// TIA Portal V20 export
FUNCTION "Map01" : Void   // FC126, LAD
// stored: Namespace Unit1, SetENOAutomatically false
   VAR_TEMP   // added for the SCL form of the ladder/FBD networks
      _w1 : Bool;
   END_VAR
BEGIN

REGION Network 1: Autocycle Running
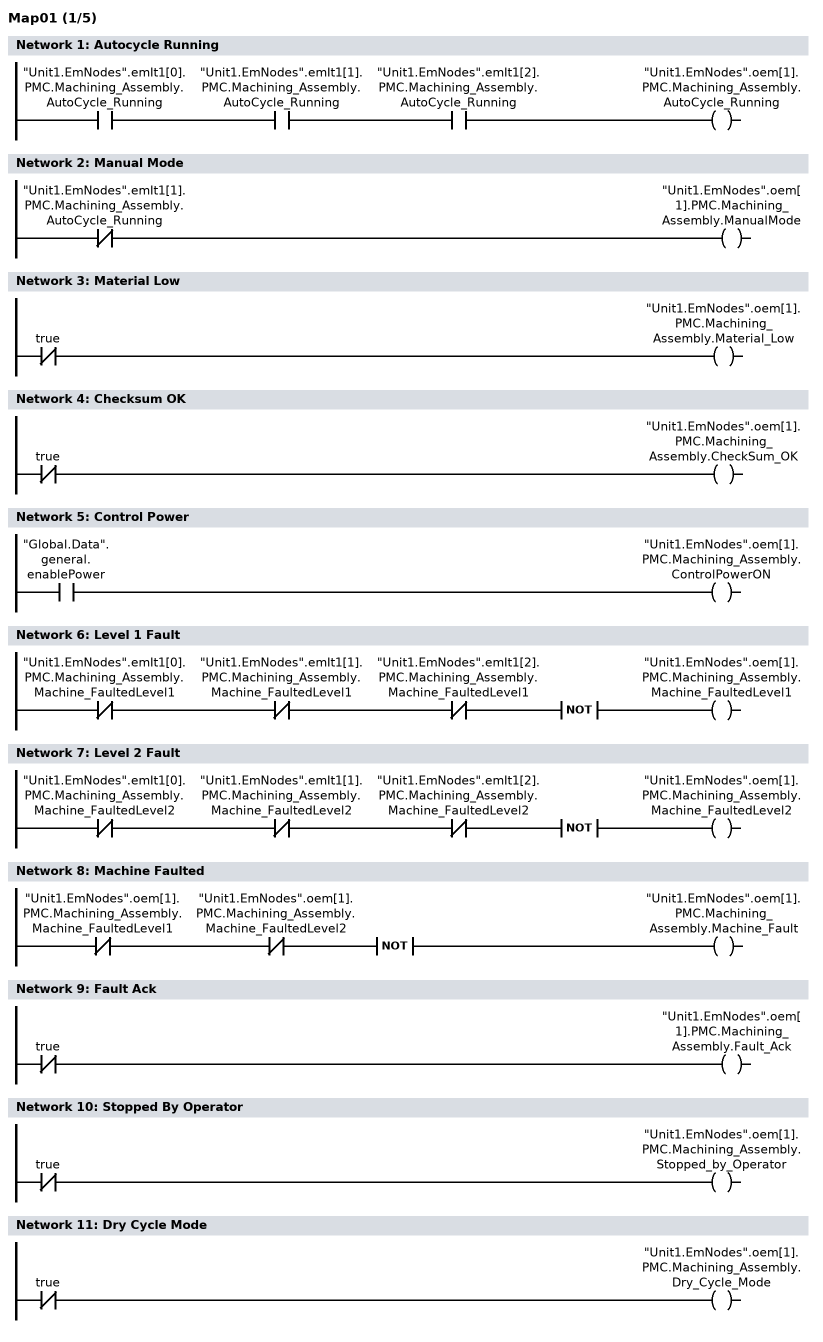
   RUNG wire#powerrail
      Contact( "Unit1.EmNodes".emIt1[0].PMC.Machining_Assembly.AutoCycle_Running )
      Contact( "Unit1.EmNodes".emIt1[1].PMC.Machining_Assembly.AutoCycle_Running )
      Contact( "Unit1.EmNodes".emIt1[2].PMC.Machining_Assembly.AutoCycle_Running )
      Coil( "Unit1.EmNodes".oem[1].PMC.Machining_Assembly.AutoCycle_Running )
   END_RUNG
   // the same network as SCL:
   "Unit1.EmNodes".oem[1].PMC.Machining_Assembly.AutoCycle_Running := "Unit1.EmNodes".emIt1[0].PMC.Machining_Assembly.AutoCycle_Running AND "Unit1.EmNodes".emIt1[1].PMC.Machining_Assembly.AutoCycle_Running AND "Unit1.EmNodes".emIt1[2].PMC.Machining_Assembly.AutoCycle_Running;
END_REGION

REGION Network 2: Manual Mode
   RUNG wire#powerrail
      I_Contact( "Unit1.EmNodes".emIt1[1].PMC.Machining_Assembly.AutoCycle_Running )
      Coil( "Unit1.EmNodes".oem[1].PMC.Machining_Assembly.ManualMode )
   END_RUNG
   // the same network as SCL:
   "Unit1.EmNodes".oem[1].PMC.Machining_Assembly.ManualMode := NOT "Unit1.EmNodes".emIt1[1].PMC.Machining_Assembly.AutoCycle_Running;
END_REGION

REGION Network 3: Material Low
   RUNG wire#powerrail
      I_Contact( true )
      Coil( "Unit1.EmNodes".oem[1].PMC.Machining_Assembly.Material_Low )
   END_RUNG
   // the same network as SCL:
   "Unit1.EmNodes".oem[1].PMC.Machining_Assembly.Material_Low := NOT true;
END_REGION

REGION Network 4: Checksum OK
   RUNG wire#powerrail
      I_Contact( true )
      Coil( "Unit1.EmNodes".oem[1].PMC.Machining_Assembly.CheckSum_OK )
   END_RUNG
   // the same network as SCL:
   "Unit1.EmNodes".oem[1].PMC.Machining_Assembly.CheckSum_OK := NOT true;
END_REGION

REGION Network 5: Control Power
   RUNG wire#powerrail
      Contact( "Global.Data".general.enablePower )
      Coil( "Unit1.EmNodes".oem[1].PMC.Machining_Assembly.ControlPowerON )
   END_RUNG
   // the same network as SCL:
   "Unit1.EmNodes".oem[1].PMC.Machining_Assembly.ControlPowerON := "Global.Data".general.enablePower;
END_REGION

REGION Network 6: Level 1 Fault
   RUNG wire#powerrail
      I_Contact( "Unit1.EmNodes".emIt1[0].PMC.Machining_Assembly.Machine_FaultedLevel1 )
      I_Contact( "Unit1.EmNodes".emIt1[1].PMC.Machining_Assembly.Machine_FaultedLevel1 )
      I_Contact( "Unit1.EmNodes".emIt1[2].PMC.Machining_Assembly.Machine_FaultedLevel1 )
      Not()
      Coil( "Unit1.EmNodes".oem[1].PMC.Machining_Assembly.Machine_FaultedLevel1 )
   END_RUNG
   // the same network as SCL:
   "Unit1.EmNodes".oem[1].PMC.Machining_Assembly.Machine_FaultedLevel1 := NOT (NOT "Unit1.EmNodes".emIt1[0].PMC.Machining_Assembly.Machine_FaultedLevel1 AND NOT "Unit1.EmNodes".emIt1[1].PMC.Machining_Assembly.Machine_FaultedLevel1 AND NOT "Unit1.EmNodes".emIt1[2].PMC.Machining_Assembly.Machine_FaultedLevel1);
END_REGION

REGION Network 7: Level 2 Fault
   RUNG wire#powerrail
      I_Contact( "Unit1.EmNodes".emIt1[0].PMC.Machining_Assembly.Machine_FaultedLevel2 )
      I_Contact( "Unit1.EmNodes".emIt1[1].PMC.Machining_Assembly.Machine_FaultedLevel2 )
      I_Contact( "Unit1.EmNodes".emIt1[2].PMC.Machining_Assembly.Machine_FaultedLevel2 )
      Not()
      Coil( "Unit1.EmNodes".oem[1].PMC.Machining_Assembly.Machine_FaultedLevel2 )
   END_RUNG
   // the same network as SCL:
   "Unit1.EmNodes".oem[1].PMC.Machining_Assembly.Machine_FaultedLevel2 := NOT (NOT "Unit1.EmNodes".emIt1[0].PMC.Machining_Assembly.Machine_FaultedLevel2 AND NOT "Unit1.EmNodes".emIt1[1].PMC.Machining_Assembly.Machine_FaultedLevel2 AND NOT "Unit1.EmNodes".emIt1[2].PMC.Machining_Assembly.Machine_FaultedLevel2);
END_REGION

REGION Network 8: Machine Faulted
   RUNG wire#powerrail
      I_Contact( "Unit1.EmNodes".oem[1].PMC.Machining_Assembly.Machine_FaultedLevel1 )
      I_Contact( "Unit1.EmNodes".oem[1].PMC.Machining_Assembly.Machine_FaultedLevel2 )
      Not()
      Coil( "Unit1.EmNodes".oem[1].PMC.Machining_Assembly.Machine_Fault )
   END_RUNG
   // the same network as SCL:
   "Unit1.EmNodes".oem[1].PMC.Machining_Assembly.Machine_Fault := NOT (NOT "Unit1.EmNodes".oem[1].PMC.Machining_Assembly.Machine_FaultedLevel1 AND NOT "Unit1.EmNodes".oem[1].PMC.Machining_Assembly.Machine_FaultedLevel2);
END_REGION

REGION Network 9: Fault Ack
   RUNG wire#powerrail
      I_Contact( true )
      Coil( "Unit1.EmNodes".oem[1].PMC.Machining_Assembly.Fault_Ack )
   END_RUNG
   // the same network as SCL:
   "Unit1.EmNodes".oem[1].PMC.Machining_Assembly.Fault_Ack := NOT true;
END_REGION

REGION Network 10: Stopped By Operator
   RUNG wire#powerrail
      I_Contact( true )
      Coil( "Unit1.EmNodes".oem[1].PMC.Machining_Assembly.Stopped_by_Operator )
   END_RUNG
   // the same network as SCL:
   "Unit1.EmNodes".oem[1].PMC.Machining_Assembly.Stopped_by_Operator := NOT true;
END_REGION

REGION Network 11: Dry Cycle Mode
   RUNG wire#powerrail
      I_Contact( true )
      Coil( "Unit1.EmNodes".oem[1].PMC.Machining_Assembly.Dry_Cycle_Mode )
   END_RUNG
   // the same network as SCL:
   "Unit1.EmNodes".oem[1].PMC.Machining_Assembly.Dry_Cycle_Mode := NOT true;
END_REGION

REGION Network 12: Blocked
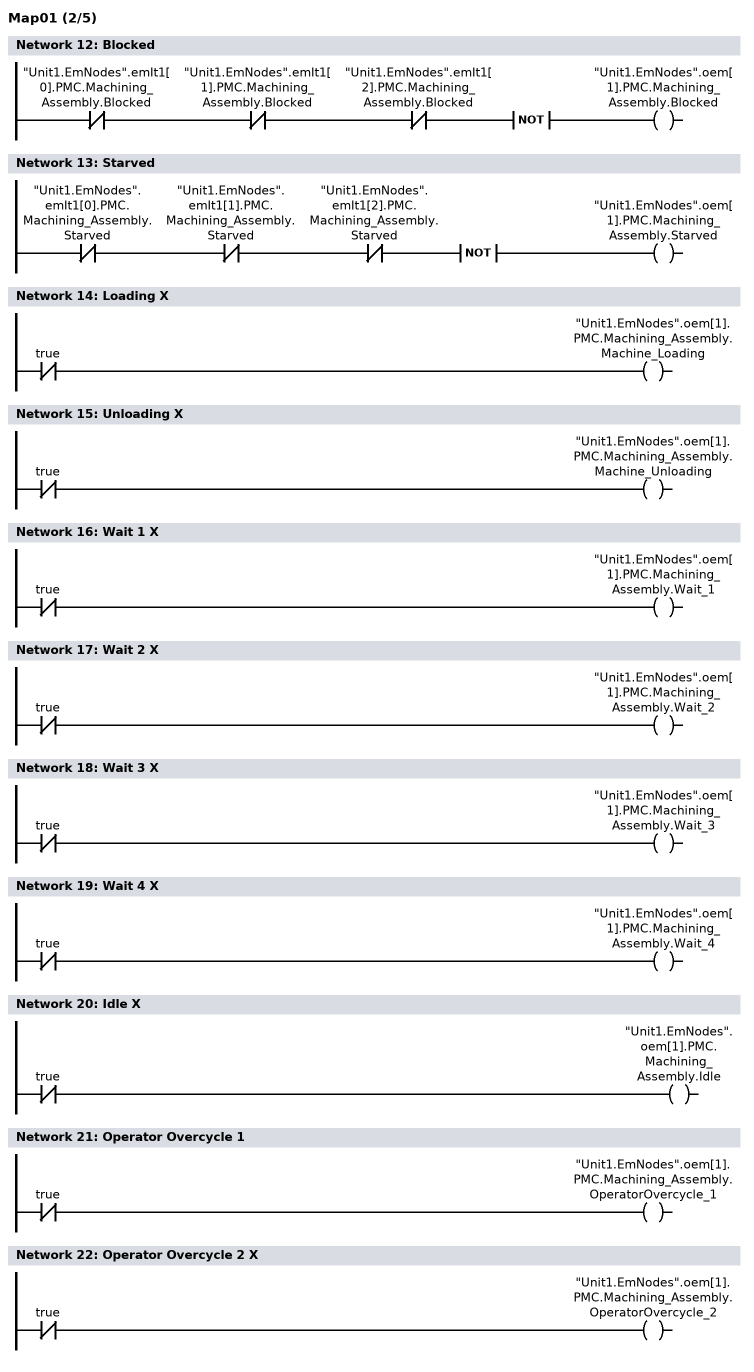
   RUNG wire#powerrail
      I_Contact( "Unit1.EmNodes".emIt1[0].PMC.Machining_Assembly.Blocked )
      I_Contact( "Unit1.EmNodes".emIt1[1].PMC.Machining_Assembly.Blocked )
      I_Contact( "Unit1.EmNodes".emIt1[2].PMC.Machining_Assembly.Blocked )
      Not()
      Coil( "Unit1.EmNodes".oem[1].PMC.Machining_Assembly.Blocked )
   END_RUNG
   // the same network as SCL:
   "Unit1.EmNodes".oem[1].PMC.Machining_Assembly.Blocked := NOT (NOT "Unit1.EmNodes".emIt1[0].PMC.Machining_Assembly.Blocked AND NOT "Unit1.EmNodes".emIt1[1].PMC.Machining_Assembly.Blocked AND NOT "Unit1.EmNodes".emIt1[2].PMC.Machining_Assembly.Blocked);
END_REGION

REGION Network 13: Starved
   RUNG wire#powerrail
      I_Contact( "Unit1.EmNodes".emIt1[0].PMC.Machining_Assembly.Starved )
      I_Contact( "Unit1.EmNodes".emIt1[1].PMC.Machining_Assembly.Starved )
      I_Contact( "Unit1.EmNodes".emIt1[2].PMC.Machining_Assembly.Starved )
      Not()
      Coil( "Unit1.EmNodes".oem[1].PMC.Machining_Assembly.Starved )
   END_RUNG
   // the same network as SCL:
   "Unit1.EmNodes".oem[1].PMC.Machining_Assembly.Starved := NOT (NOT "Unit1.EmNodes".emIt1[0].PMC.Machining_Assembly.Starved AND NOT "Unit1.EmNodes".emIt1[1].PMC.Machining_Assembly.Starved AND NOT "Unit1.EmNodes".emIt1[2].PMC.Machining_Assembly.Starved);
END_REGION

REGION Network 14: Loading X
   RUNG wire#powerrail
      I_Contact( true )
      Coil( "Unit1.EmNodes".oem[1].PMC.Machining_Assembly.Machine_Loading )
   END_RUNG
   // the same network as SCL:
   "Unit1.EmNodes".oem[1].PMC.Machining_Assembly.Machine_Loading := NOT true;
END_REGION

REGION Network 15: Unloading X
   RUNG wire#powerrail
      I_Contact( true )
      Coil( "Unit1.EmNodes".oem[1].PMC.Machining_Assembly.Machine_Unloading )
   END_RUNG
   // the same network as SCL:
   "Unit1.EmNodes".oem[1].PMC.Machining_Assembly.Machine_Unloading := NOT true;
END_REGION

REGION Network 16: Wait 1 X
   RUNG wire#powerrail
      I_Contact( true )
      Coil( "Unit1.EmNodes".oem[1].PMC.Machining_Assembly.Wait_1 )
   END_RUNG
   // the same network as SCL:
   "Unit1.EmNodes".oem[1].PMC.Machining_Assembly.Wait_1 := NOT true;
END_REGION

REGION Network 17: Wait 2 X
   RUNG wire#powerrail
      I_Contact( true )
      Coil( "Unit1.EmNodes".oem[1].PMC.Machining_Assembly.Wait_2 )
   END_RUNG
   // the same network as SCL:
   "Unit1.EmNodes".oem[1].PMC.Machining_Assembly.Wait_2 := NOT true;
END_REGION

REGION Network 18: Wait 3 X
   RUNG wire#powerrail
      I_Contact( true )
      Coil( "Unit1.EmNodes".oem[1].PMC.Machining_Assembly.Wait_3 )
   END_RUNG
   // the same network as SCL:
   "Unit1.EmNodes".oem[1].PMC.Machining_Assembly.Wait_3 := NOT true;
END_REGION

REGION Network 19: Wait 4 X
   RUNG wire#powerrail
      I_Contact( true )
      Coil( "Unit1.EmNodes".oem[1].PMC.Machining_Assembly.Wait_4 )
   END_RUNG
   // the same network as SCL:
   "Unit1.EmNodes".oem[1].PMC.Machining_Assembly.Wait_4 := NOT true;
END_REGION

REGION Network 20: Idle X
   RUNG wire#powerrail
      I_Contact( true )
      Coil( "Unit1.EmNodes".oem[1].PMC.Machining_Assembly.Idle )
   END_RUNG
   // the same network as SCL:
   "Unit1.EmNodes".oem[1].PMC.Machining_Assembly.Idle := NOT true;
END_REGION

REGION Network 21: Operator Overcycle 1
   RUNG wire#powerrail
      I_Contact( true )
      Coil( "Unit1.EmNodes".oem[1].PMC.Machining_Assembly.OperatorOvercycle_1 )
   END_RUNG
   // the same network as SCL:
   "Unit1.EmNodes".oem[1].PMC.Machining_Assembly.OperatorOvercycle_1 := NOT true;
END_REGION

REGION Network 22: Operator Overcycle 2 X
   RUNG wire#powerrail
      I_Contact( true )
      Coil( "Unit1.EmNodes".oem[1].PMC.Machining_Assembly.OperatorOvercycle_2 )
   END_RUNG
   // the same network as SCL:
   "Unit1.EmNodes".oem[1].PMC.Machining_Assembly.OperatorOvercycle_2 := NOT true;
END_REGION

REGION Network 23: Operator Overcycle 3 X
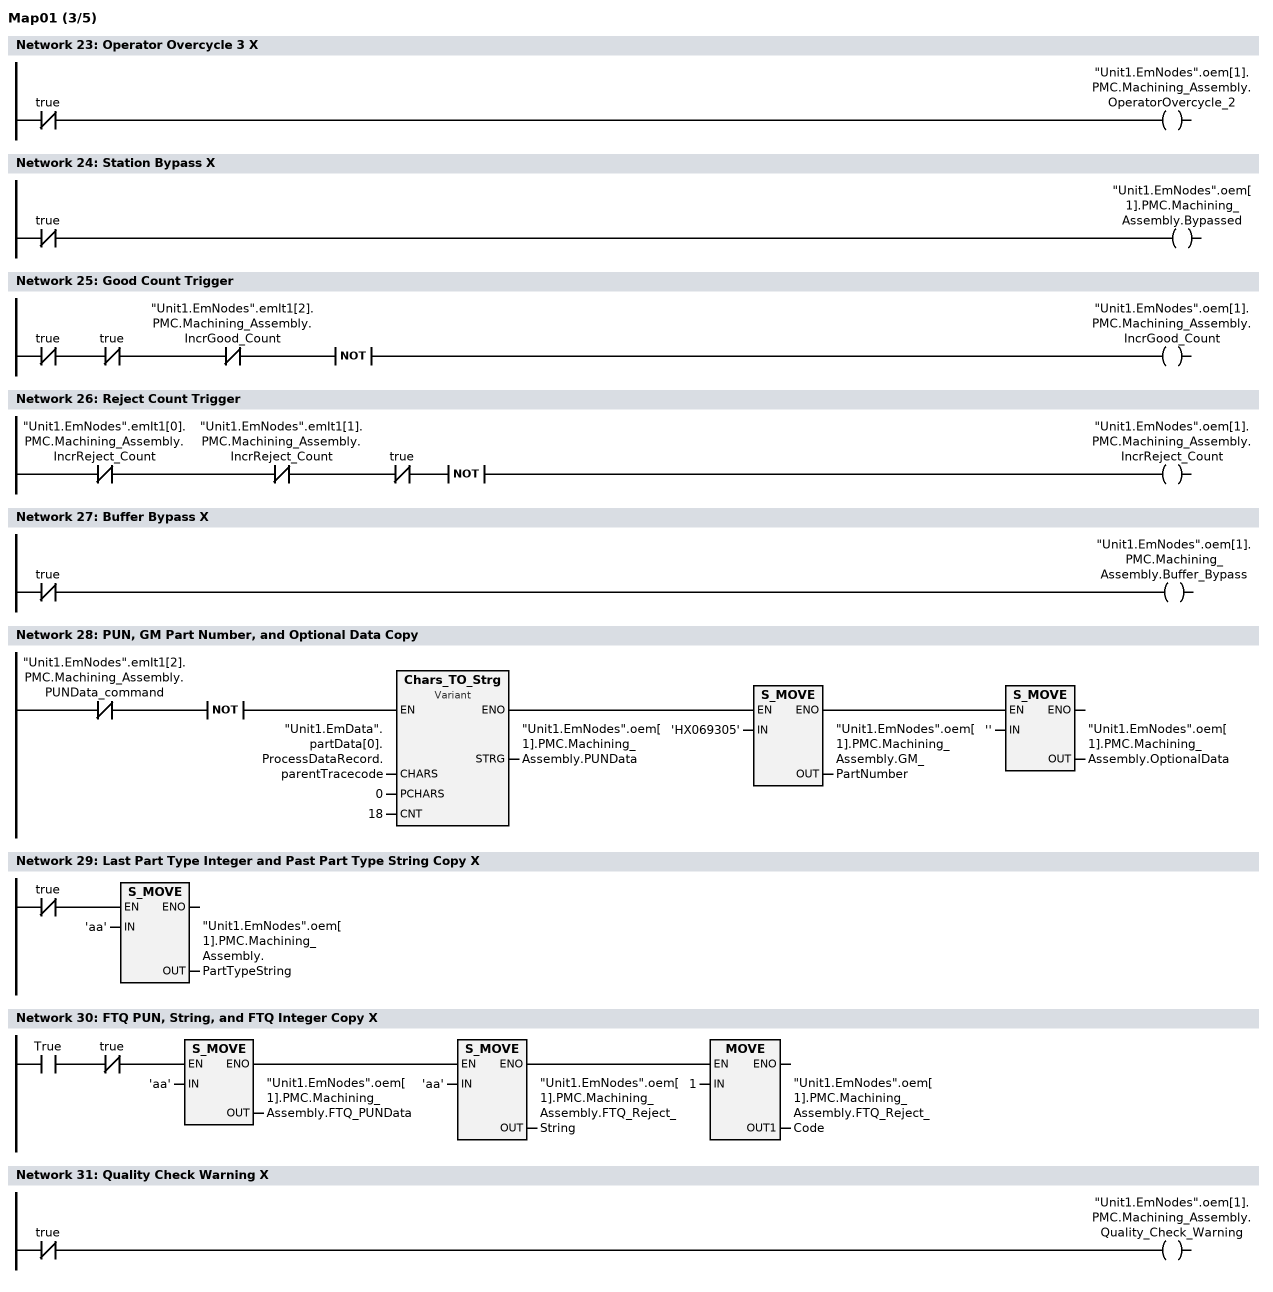
   RUNG wire#powerrail
      I_Contact( true )
      Coil( "Unit1.EmNodes".oem[1].PMC.Machining_Assembly.OperatorOvercycle_2 )
   END_RUNG
   // the same network as SCL:
   "Unit1.EmNodes".oem[1].PMC.Machining_Assembly.OperatorOvercycle_2 := NOT true;
END_REGION

REGION Network 24: Station Bypass X
   RUNG wire#powerrail
      I_Contact( true )
      Coil( "Unit1.EmNodes".oem[1].PMC.Machining_Assembly.Bypassed )
   END_RUNG
   // the same network as SCL:
   "Unit1.EmNodes".oem[1].PMC.Machining_Assembly.Bypassed := NOT true;
END_REGION

REGION Network 25: Good Count Trigger
   RUNG wire#powerrail
      I_Contact( true )
      I_Contact( true )
      I_Contact( "Unit1.EmNodes".emIt1[2].PMC.Machining_Assembly.IncrGood_Count )
      Not()
      Coil( "Unit1.EmNodes".oem[1].PMC.Machining_Assembly.IncrGood_Count )
   END_RUNG
   // the same network as SCL:
   "Unit1.EmNodes".oem[1].PMC.Machining_Assembly.IncrGood_Count := NOT (NOT true AND NOT true AND NOT "Unit1.EmNodes".emIt1[2].PMC.Machining_Assembly.IncrGood_Count);
END_REGION

REGION Network 26: Reject Count Trigger
   RUNG wire#powerrail
      I_Contact( "Unit1.EmNodes".emIt1[0].PMC.Machining_Assembly.IncrReject_Count )
      I_Contact( "Unit1.EmNodes".emIt1[1].PMC.Machining_Assembly.IncrReject_Count )
      I_Contact( true )
      Not()
      Coil( "Unit1.EmNodes".oem[1].PMC.Machining_Assembly.IncrReject_Count )
   END_RUNG
   // the same network as SCL:
   "Unit1.EmNodes".oem[1].PMC.Machining_Assembly.IncrReject_Count := NOT (NOT "Unit1.EmNodes".emIt1[0].PMC.Machining_Assembly.IncrReject_Count AND NOT "Unit1.EmNodes".emIt1[1].PMC.Machining_Assembly.IncrReject_Count AND NOT true);
END_REGION

REGION Network 27: Buffer Bypass X
   RUNG wire#powerrail
      I_Contact( true )
      Coil( "Unit1.EmNodes".oem[1].PMC.Machining_Assembly.Buffer_Bypass )
   END_RUNG
   // the same network as SCL:
   "Unit1.EmNodes".oem[1].PMC.Machining_Assembly.Buffer_Bypass := NOT true;
END_REGION

REGION Network 28: PUN, GM Part Number, and Optional Data Copy
   RUNG wire#powerrail
      I_Contact( "Unit1.EmNodes".emIt1[2].PMC.Machining_Assembly.PUNData_command )
      Not()
      { S7_Templates := "[ptr_type := Variant, str_type := String]" } Chars_TO_Strg(Chars := "Unit1.EmData".partData[0].ProcessDataRecord.parentTracecode, pChars := 0, Cnt := 18, Strg => "Unit1.EmNodes".oem[1].PMC.Machining_Assembly.PUNData)
      S_Move(in := 'HX069305', out => "Unit1.EmNodes".oem[1].PMC.Machining_Assembly.GM_PartNumber)
      S_Move(in := '', out => "Unit1.EmNodes".oem[1].PMC.Machining_Assembly.OptionalData)
   END_RUNG
   // the same network as SCL:
   Chars_TO_Strg(EN := NOT (NOT "Unit1.EmNodes".emIt1[2].PMC.Machining_Assembly.PUNData_command),
                 Chars := "Unit1.EmData".partData[0].ProcessDataRecord.parentTracecode,
                 pChars := 0,
                 Cnt := 18,
                 Strg => "Unit1.EmNodes".oem[1].PMC.Machining_Assembly.PUNData,
                 ENO => #_w1);
   IF #_w1 THEN
       "Unit1.EmNodes".oem[1].PMC.Machining_Assembly.GM_PartNumber := 'HX069305';
       "Unit1.EmNodes".oem[1].PMC.Machining_Assembly.OptionalData := '';
   END_IF;
END_REGION

REGION Network 29: Last Part Type Integer and Past Part Type String Copy X
   RUNG wire#powerrail
      I_Contact( true )
      S_Move(in := 'aa', out => "Unit1.EmNodes".oem[1].PMC.Machining_Assembly.PartTypeString)
   END_RUNG
   // the same network as SCL:
   IF NOT true THEN "Unit1.EmNodes".oem[1].PMC.Machining_Assembly.PartTypeString := 'aa'; END_IF;
END_REGION

REGION Network 30: FTQ PUN, String, and FTQ Integer Copy X
   RUNG wire#powerrail
      Contact( True )
      I_Contact( true )
      S_Move(in := 'aa', out => "Unit1.EmNodes".oem[1].PMC.Machining_Assembly.FTQ_PUNData)
      S_Move(in := 'aa', out => "Unit1.EmNodes".oem[1].PMC.Machining_Assembly.FTQ_Reject_String)
      Move(in := 1, out1 => "Unit1.EmNodes".oem[1].PMC.Machining_Assembly.FTQ_Reject_Code)
   END_RUNG
   // the same network as SCL:
   IF True AND NOT true THEN
       "Unit1.EmNodes".oem[1].PMC.Machining_Assembly.FTQ_PUNData := 'aa';
       "Unit1.EmNodes".oem[1].PMC.Machining_Assembly.FTQ_Reject_String := 'aa';
       "Unit1.EmNodes".oem[1].PMC.Machining_Assembly.FTQ_Reject_Code := 1;
   END_IF;
END_REGION

REGION Network 31: Quality Check Warning X
   RUNG wire#powerrail
      I_Contact( true )
      Coil( "Unit1.EmNodes".oem[1].PMC.Machining_Assembly.Quality_Check_Warning )
   END_RUNG
   // the same network as SCL:
   "Unit1.EmNodes".oem[1].PMC.Machining_Assembly.Quality_Check_Warning := NOT true;
END_REGION

REGION Network 32: Quality Check Fault X
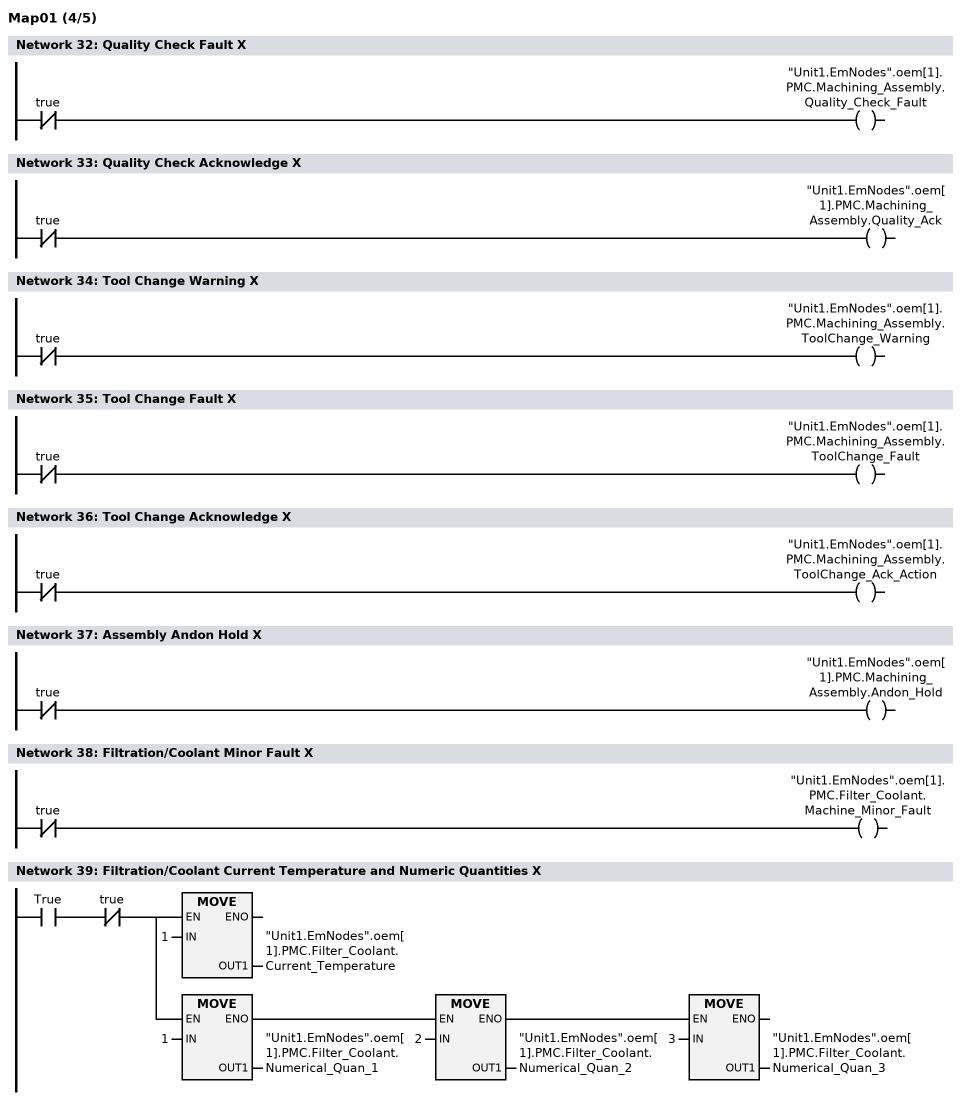
   RUNG wire#powerrail
      I_Contact( true )
      Coil( "Unit1.EmNodes".oem[1].PMC.Machining_Assembly.Quality_Check_Fault )
   END_RUNG
   // the same network as SCL:
   "Unit1.EmNodes".oem[1].PMC.Machining_Assembly.Quality_Check_Fault := NOT true;
END_REGION

REGION Network 33: Quality Check Acknowledge X
   RUNG wire#powerrail
      I_Contact( true )
      Coil( "Unit1.EmNodes".oem[1].PMC.Machining_Assembly.Quality_Ack )
   END_RUNG
   // the same network as SCL:
   "Unit1.EmNodes".oem[1].PMC.Machining_Assembly.Quality_Ack := NOT true;
END_REGION

REGION Network 34: Tool Change Warning X
   RUNG wire#powerrail
      I_Contact( true )
      Coil( "Unit1.EmNodes".oem[1].PMC.Machining_Assembly.ToolChange_Warning )
   END_RUNG
   // the same network as SCL:
   "Unit1.EmNodes".oem[1].PMC.Machining_Assembly.ToolChange_Warning := NOT true;
END_REGION

REGION Network 35: Tool Change Fault X
   RUNG wire#powerrail
      I_Contact( true )
      Coil( "Unit1.EmNodes".oem[1].PMC.Machining_Assembly.ToolChange_Fault )
   END_RUNG
   // the same network as SCL:
   "Unit1.EmNodes".oem[1].PMC.Machining_Assembly.ToolChange_Fault := NOT true;
END_REGION

REGION Network 36: Tool Change Acknowledge X
   RUNG wire#powerrail
      I_Contact( true )
      Coil( "Unit1.EmNodes".oem[1].PMC.Machining_Assembly.ToolChange_Ack_Action )
   END_RUNG
   // the same network as SCL:
   "Unit1.EmNodes".oem[1].PMC.Machining_Assembly.ToolChange_Ack_Action := NOT true;
END_REGION

REGION Network 37: Assembly Andon Hold X
   RUNG wire#powerrail
      I_Contact( true )
      Coil( "Unit1.EmNodes".oem[1].PMC.Machining_Assembly.Andon_Hold )
   END_RUNG
   // the same network as SCL:
   "Unit1.EmNodes".oem[1].PMC.Machining_Assembly.Andon_Hold := NOT true;
END_REGION

REGION Network 38: Filtration/Coolant Minor Fault X
   RUNG wire#powerrail
      I_Contact( true )
      Coil( "Unit1.EmNodes".oem[1].PMC.Filter_Coolant.Machine_Minor_Fault )
   END_RUNG
   // the same network as SCL:
   "Unit1.EmNodes".oem[1].PMC.Filter_Coolant.Machine_Minor_Fault := NOT true;
END_REGION

REGION Network 39: Filtration/Coolant Current Temperature and Numeric Quantities X
   RUNG wire#powerrail
      Contact( True )
      I_Contact( true )
      wire#w1
      Move(in := 1, out1 => "Unit1.EmNodes".oem[1].PMC.Filter_Coolant.Current_Temperature)
   END_RUNG
   RUNG wire#w1
      Move(in := 1, out1 => "Unit1.EmNodes".oem[1].PMC.Filter_Coolant.Numerical_Quan_1)
      Move(in := 2, out1 => "Unit1.EmNodes".oem[1].PMC.Filter_Coolant.Numerical_Quan_2)
      Move(in := 3, out1 => "Unit1.EmNodes".oem[1].PMC.Filter_Coolant.Numerical_Quan_3)
   END_RUNG
   // the same network as SCL:
   IF True AND NOT true THEN
       "Unit1.EmNodes".oem[1].PMC.Filter_Coolant.Current_Temperature := 1;
       "Unit1.EmNodes".oem[1].PMC.Filter_Coolant.Numerical_Quan_1 := 1;
       "Unit1.EmNodes".oem[1].PMC.Filter_Coolant.Numerical_Quan_2 := 2;
       "Unit1.EmNodes".oem[1].PMC.Filter_Coolant.Numerical_Quan_3 := 3;
   END_IF;
END_REGION

REGION Network 40: Filtration/Coolant Tank Level Data X
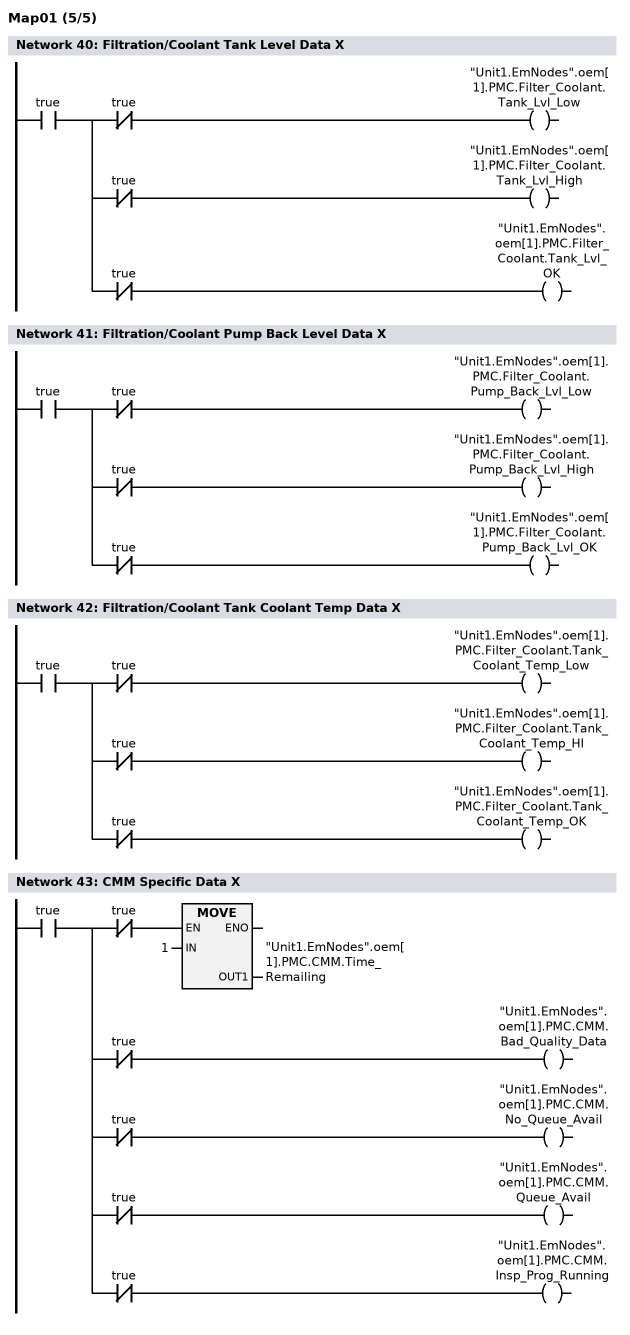
   RUNG wire#powerrail
      Contact( true )
      wire#w1
      I_Contact( true )
      Coil( "Unit1.EmNodes".oem[1].PMC.Filter_Coolant.Tank_Lvl_Low )
   END_RUNG
   RUNG wire#w1
      I_Contact( true )
      Coil( "Unit1.EmNodes".oem[1].PMC.Filter_Coolant.Tank_Lvl_High )
   END_RUNG
   RUNG wire#w1
      I_Contact( true )
      Coil( "Unit1.EmNodes".oem[1].PMC.Filter_Coolant.Tank_Lvl_OK )
   END_RUNG
   // the same network as SCL:
   "Unit1.EmNodes".oem[1].PMC.Filter_Coolant.Tank_Lvl_Low := true AND NOT true;
   "Unit1.EmNodes".oem[1].PMC.Filter_Coolant.Tank_Lvl_High := true AND NOT true;
   "Unit1.EmNodes".oem[1].PMC.Filter_Coolant.Tank_Lvl_OK := true AND NOT true;
END_REGION

REGION Network 41: Filtration/Coolant Pump Back Level Data X
   RUNG wire#powerrail
      Contact( true )
      wire#w1
      I_Contact( true )
      Coil( "Unit1.EmNodes".oem[1].PMC.Filter_Coolant.Pump_Back_Lvl_Low )
   END_RUNG
   RUNG wire#w1
      I_Contact( true )
      Coil( "Unit1.EmNodes".oem[1].PMC.Filter_Coolant.Pump_Back_Lvl_High )
   END_RUNG
   RUNG wire#w1
      I_Contact( true )
      Coil( "Unit1.EmNodes".oem[1].PMC.Filter_Coolant.Pump_Back_Lvl_OK )
   END_RUNG
   // the same network as SCL:
   "Unit1.EmNodes".oem[1].PMC.Filter_Coolant.Pump_Back_Lvl_Low := true AND NOT true;
   "Unit1.EmNodes".oem[1].PMC.Filter_Coolant.Pump_Back_Lvl_High := true AND NOT true;
   "Unit1.EmNodes".oem[1].PMC.Filter_Coolant.Pump_Back_Lvl_OK := true AND NOT true;
END_REGION

REGION Network 42: Filtration/Coolant Tank Coolant Temp Data X
   RUNG wire#powerrail
      Contact( true )
      wire#w1
      I_Contact( true )
      Coil( "Unit1.EmNodes".oem[1].PMC.Filter_Coolant.Tank_Coolant_Temp_Low )
   END_RUNG
   RUNG wire#w1
      I_Contact( true )
      Coil( "Unit1.EmNodes".oem[1].PMC.Filter_Coolant.Tank_Coolant_Temp_HI )
   END_RUNG
   RUNG wire#w1
      I_Contact( true )
      Coil( "Unit1.EmNodes".oem[1].PMC.Filter_Coolant.Tank_Coolant_Temp_OK )
   END_RUNG
   // the same network as SCL:
   "Unit1.EmNodes".oem[1].PMC.Filter_Coolant.Tank_Coolant_Temp_Low := true AND NOT true;
   "Unit1.EmNodes".oem[1].PMC.Filter_Coolant.Tank_Coolant_Temp_HI := true AND NOT true;
   "Unit1.EmNodes".oem[1].PMC.Filter_Coolant.Tank_Coolant_Temp_OK := true AND NOT true;
END_REGION

REGION Network 43: CMM Specific Data X
   RUNG wire#powerrail
      Contact( true )
      wire#w1
      I_Contact( true )
      Move(in := 1, out1 => "Unit1.EmNodes".oem[1].PMC.CMM.Time_Remailing)
   END_RUNG
   RUNG wire#w1
      I_Contact( true )
      Coil( "Unit1.EmNodes".oem[1].PMC.CMM.Bad_Quality_Data )
   END_RUNG
   RUNG wire#w1
      I_Contact( true )
      Coil( "Unit1.EmNodes".oem[1].PMC.CMM.No_Queue_Avail )
   END_RUNG
   RUNG wire#w1
      I_Contact( true )
      Coil( "Unit1.EmNodes".oem[1].PMC.CMM.Queue_Avail )
   END_RUNG
   RUNG wire#w1
      I_Contact( true )
      Coil( "Unit1.EmNodes".oem[1].PMC.CMM.Insp_Prog_Running )
   END_RUNG
   // the same network as SCL:
   IF true AND NOT true THEN "Unit1.EmNodes".oem[1].PMC.CMM.Time_Remailing := 1; END_IF;
   "Unit1.EmNodes".oem[1].PMC.CMM.Bad_Quality_Data := true AND NOT true;
   "Unit1.EmNodes".oem[1].PMC.CMM.No_Queue_Avail := true AND NOT true;
   "Unit1.EmNodes".oem[1].PMC.CMM.Queue_Avail := true AND NOT true;
   "Unit1.EmNodes".oem[1].PMC.CMM.Insp_Prog_Running := true AND NOT true;
END_REGION
END_FUNCTION
